VAR_GLOBAL
	//AXIS_1 : UINT := 1;
	//AXIS_2 : UINT := 2;
END_VAR

(* stored: Version 1.1.0.1, ProductVersion 3.1.4024.11
   GVL GVL_AxisNames: Id {ac2d037b-2b8c-41f4-8d85-bcb635f10da5} *)
